FUNCTION_BLOCK DIVIDE (* Basic Function Block Type *)
  (* Standard: 61499-2 *)
  (* Version 0.0, 7/8/2026, Schneider Electric, Template *)
  PACKAGE SE.Nereda;
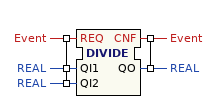
  EVENT_INPUT
    REQ WITH QI1, QI2; (* Normal Execution Request *)
  END_EVENT
  EVENT_OUTPUT
    CNF WITH QO; (* Execution Confirmation *)
  END_EVENT
  VAR_INPUT
    QI1 : REAL; (* Input event qualifier *)
    QI2 : REAL;
  END_VAR
  VAR_OUTPUT
    QO : REAL; (* Output event qualifier *)
  END_VAR
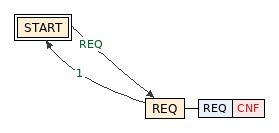
  EC_STATES
    START; (* Initial State *)
    REQ : REQ -> CNF; (* Normal execution *)
  END_STATES
  EC_TRANSITIONS
    START TO REQ := REQ;
    REQ TO START := 1;
  END_TRANSITIONS
  ALGORITHM REQ IN ST: (* Normally executed algorithm *)
;
QO := QI1 / QI2;
  END_ALGORITHM
END_FUNCTION_BLOCK
